        if issues_value == -2 and direction_changes < 2:
			#target unreachable
            if rotation_direction == "pos":
                rotation_direction = "neg"
                direction_changes += 1
                r = -1 #rotation factor to make the rotation negative
            else:
                rotation_direction = "pos"
                direction_changes += 1
                r = 1 #rotation factor to make the rotation positive
            issues_value, target_new_pose = test_issues_point(target, r*rotation_step)
            target.setPose(target_new_pose)

        elif issues_value > 0 and rep < repmax:
			#collision
            RDK.setCollisionActive(COLLISION_OFF)
            if DEBUG:
                is_active = RDK.Command("CollisionActive")
                print(f"collsion active? should be off (0) {is_active}")
                debuglist.append(f"collsion active? should be off (0) {is_active}")

            ROBOT.MoveJ(target.Pose())
            if rotation_direction == "neg":
                r = -1
            elif rotation_direction == "pos":
                r = 1
            issues_value, target_new_pose = test_issues_point(target, r*rotation_step)
            target.setPose(target_new_pose)
            rep += 1

        elif direction_changes >= 2 or rep >= repmax:
            break

        else:
            RDK.ShowMessage(f"Unknown error occured at Hole {idx} while looking for collision free position")
            if DEBUG:
                print(f"Unknown error occured at Hole {idx} while looking for collision free position")
                debuglist.append(f"Unknown error occured at Hole {idx} while looking for collision free position")

    direction_changes = 0
    if issues_value == 0:
        print(f"No issues at Hole {idx}")
        debuglist.append(f"No issues at Hole {idx}")
    elif direction_changes >= 2 or rep >= repmax or s >= 100:
        RDK.ShowMessage(f"No solution found for Hole {idx}", False)
        holes_no_solution.append(idx)
        if DEBUG:
            print(f"No solution found for Hole {idx}")
            debuglist.append(f"No solution found for Hole {idx}")
    else:
        RDK.ShowMessage(f"Unknown error occured at Hole {idx} while looking for collision free position")
        if DEBUG:
            print(f"Unknown error occured at Hole {idx} while looking for collision free position")
            debuglist.append(f"Unknown error occured at Hole {idx} while looking for collision free position")


MAKE_GUI_PROGRAM = True

ROBOT.setFrame(FRAME)
ROBOT.setTool(TOOL)

if RDK.RunMode() == RUNMODE_SIMULATE:
    MAKE_GUI_PROGRAM = True
    # MAKE_GUI_PROGRAM = mbox('Do you want to create a new program? If not, the robot will just move along the targets', 'Yes', 'No')
else:
    # if we run in program generation mode just move the robot
    MAKE_GUI_PROGRAM = False

if MAKE_GUI_PROGRAM:
    RDK.Render(False)  # Faster if we turn render off
    make_targets(csv_file)
else:
    l

RDK.ShowMessage(f"Holes without solution: {holes_no_solution}")

if DEBUG:
    print(f"Holes without solution: {holes_no_solution}")
    debuglist.append(f"Holes without solution: {holes_no_solution}")

    current_time = datetime.datetime.now()
    filename = os.path.splitext(os.path.basename(__file__))
    with open("C:/Users/Laura/Documents/1.Windesheim/Stage/2024/Lectoraat/Deelvragen/2.Targets maken/debugfile.txt", "a") as file:
        file.write("\n\n-----------------------------------------------\n")
        file.write(current_time.strftime("%c"))
        file.write("\n-----------------------------------------------\n")
        for prints in debuglist:
            file.write(prints)
            file.write("\n")
        file.write(holes_no_solution)
        file.write(filename[0])

--- Python program Addmoveshanktoprog ---
from robodk import robolink, robomath

# Connect to RoboDK
RDK = robolink.Robolink()

# Ask the user to select the program to duplicate
orig_prog = RDK.ItemUserPick("Select the program to duplicate", robolink.ITEM_TYPE_PROGRAM)
if not orig_prog.Valid():
    print("No valid program selected.")
    quit()

# Create a new program (a duplicate) with a new name
new_prog_name = "New_" + orig_prog.Name()
new_prog = RDK.AddProgram(new_prog_name)
print("Creating new program:", new_prog.Name())

# Get the number of instructions from the original program
ins_count = orig_prog.InstructionCount()
print("Original program '{}' has {} instructions.".format(orig_prog.Name(), ins_count))

# Iterate over each instruction in the original program
for i in range(ins_count):
    # Retrieve instruction info as a dictionary.
    # Note: Calling setParam(i) with only the index returns the instruction information.
    ins_dict = orig_prog.setParam(i)

    # Try to get the command code string from the instruction dictionary.
    # (Many instructions have a "Code" key that holds the Python command as text.)
    code_line = ins_dict.get("Code", "").strip()
    if not code_line:
        print("Skipping instruction {} because no code is available.".format(i))
        continue

    # Add the instruction to the new program
    print("Adding instruction {}: {}".format(i, code_line))
    new_prog.RunInstruction(code_line, robolink.INSTRUCTION_CALL_PROGRAM)

    # If the instruction contains "FaceTarget" then add two extra moveshank instructions after it.
    if "Face_Target" in code_line:
        print("Detected 'FaceTarget' at instruction {}. Inserting moveshank instructions.".format(i))
        new_prog.RunInstruction('move_shank(20)', robolink.INSTRUCTION_CALL_PROGRAM)
        new_prog.RunInstruction('move_shank(0)', robolink.INSTRUCTION_CALL_PROGRAM)

# Finalize the new program; this applies the modifications
new_prog.Update()
print("New program '{}' created successfully.".format(new_prog.Name()))

--- Python program importerTest ---
# This macro loads CSV target files and places them in RoboDK
# Supported CSV format: X,Y,Z,RX,RY,RZ

# Import required modules
from robodk.robolink import *  # API to communicate with RoboDK
from robodk.robomath import *  # Robot toolbox
from robodk.robodialogs import *
from robodk.robofileio import *
import robodk.robolinkutils as RDKutils

# Start communication with RoboDK
RDK = Robolink()

# Ask the user to select the robot
ROBOT = RDK.ItemUserPick('Select a robot', ITEM_TYPE_ROBOT)

# Check if the user selected a robot
if not ROBOT.Valid():
    quit()

# Get the reference frame and active tool
BASE = ROBOT.Parent()
FRAME = RDK.ItemUserPick('Reference Frame', ITEM_TYPE_FRAME)
FRAMEPOSE = RDKutils.getPoseWrt(FRAME, BASE)  # frame pose wrt robot base
TOOL = ROBOT.getLink(ITEM_TYPE_TOOL)
TOOLPOSE = RDKutils.getPoseWrt(TOOL, TOOL.Parent())  # tool pose wrt robot flange

if not FRAME.Valid() or not TOOL.Valid():
    raise Exception("Select appropriate FRAME and TOOL references")

# Function to convert XYZWPR to a pose
def xyzwpr_to_pose(xyzwpr):
    x, y, z, rx, ry, rz = xyzwpr
    return point_Zaxis_2_pose([x, y, z], [rx, ry, rz])

# Ask user to select the CSV file
csv_file = getOpenFileName(RDK.getParam('PATH_OPENSTATION'))

# Specify file codec
codec = 'utf-8'

# Load CSV target data
def load_targets(strfile):
    csvdata = LoadList(strfile, ',', codec)
    poses = []
    idxs = []
    for i in range(0, len(csvdata)):
        x, y, z, rx, ry, rz = csvdata[i][0:6]
        poses.append(xyzwpr_to_pose([x, y, z, rx, ry, rz]))
        idxs.append(i)
    return poses, idxs

# Create targets in RoboDK and move the robot to each target
def process_targets(strfile):
    poses, idxs = load_targets(strfile)
    program_name = getFileName(strfile)
    program_name = program_name.replace('-', '_').replace(' ', '_')

    # Set the robot's frame and tool
    ROBOT.setFrame(FRAME)
    ROBOT.setTool(TOOL)

    # Create a program to visit all targets
    program = RDK.AddProgram('Visit_' + program_name, ROBOT)

    for pose, idx in zip(poses, idxs):
        # Create target name
        name = 'Target-%s-%i' % (program_name, idx)

        # Delete target if it already exists
        target = RDK.Item(name, ITEM_TYPE_TARGET)
        if target.Valid():
            target.Delete()

        # Create new target
        target = RDK.AddTarget(name, FRAME, ROBOT)
        target.setPose(pose)

        # Add a movement instruction to the program
        program.MoveJ(target)

        # Optional: Move the robot to the target in simulation
        RDK.setSimulationSpeed(1)  # Normal speed
        ROBOT.MoveJ(target)

# Main execution
if __name__ == "__main__":
    # Ask user whether to just create targets or also move the robot
    move_robot = RDK.RunMode() != RUNMODE_SIMULATE

    if move_robot:
        # We're in run mode, just move the robot to targets
        poses, idxs = load_targets(csv_file)
        for pose, idx in zip(poses, idxs):
            ROBOT.MoveJ(pose)
    else:
        # We're in simulation mode, create targets and a program
        process_targets(csv_file)

    RDK.ShowMessage("Target processing complete", False)

--- program Prog20 (robot UR10e) ---
  Set Ref.: CSV Frame
  Set Tool: TCP Schroeftool at (225.74, 0.91, 101.72) mm, rotated rx 90 ry -90 rz 90 deg
  MoveL (Target 36)
  Call Program_Face_-1_0_0
  Call Program_Face_-1_0_0
  MoveL (Target 36)
  MoveL (Target 35)
  MoveJ (Target 37 new)
  MoveL (Target 37 new)
  MoveL (Target 35)
  Call Program_Face_0_-1_1
  MoveL (Target 35)
  Call Program_Face_0_-1_0
  MoveL (Target 35)

--- program Program_Face_-1_0_0 (robot UR10e) ---
  Set Ref.: CSV Frame
  Set Tool: schroevendraaier all in met meet cone (1)
  MoveL (Target 36)
  MoveL (Face_Target_-1_0_0)
  MoveL (H-12.5_30.0-9)
  MoveL (Face_Target_-1_0_0)
  MoveL (H-12.5_30.0-10)
  MoveL (Face_Target_-1_0_0)
  MoveL (H-12.5_30.0-11)
  MoveL (Face_Target_-1_0_0)
  MoveL (H-12.5_30.0-12)
  MoveL (Face_Target_-1_0_0)
  MoveL (H-12.5_30.0-13)
  MoveL (Face_Target_-1_0_0)
  MoveL (H-12.5_30.0-14)
  MoveL (Face_Target_-1_0_0)
  MoveL (H-12.5_30.0-15)
  MoveL (Face_Target_-1_0_0)
  MoveL (Target 36)

--- program Program_Face_0_0_1 (robot UR10e) ---
  Set Ref.: CSV Frame
  Set Tool: schroevendraaier all in met meet cone (1)
  MoveL (Face_Target_0_0_1)
  MoveL (H-12.4_20.0-0)
  MoveL (Face_Target_0_0_1)
  MoveL (H-12.4_20.0-1)
  MoveL (Face_Target_0_0_1)
  MoveL (H-12.4_20.0-2)
  MoveL (Face_Target_0_0_1)
  MoveL (H-12.4_20.0-3)
  MoveL (Face_Target_0_0_1)
  MoveL (H-12.4_20.0-4)
  MoveL (Face_Target_0_0_1)
  MoveL (H-12.4_20.0-5)
  MoveL (Face_Target_0_0_1)
  MoveL (H-12.4_20.0-6)
  MoveL (Face_Target_0_0_1)

--- program Program1hole3sides27May (robot UR10e) ---
  Set Ref.: CSV Frame
  Set Tool: schroevendraaier all in met meet cone (1)
  MoveL (Target 35)
  MoveL (oppak)
  Call screw_in(0)
  MoveL (Target 35)
  MoveL (Face_Target_0_-1_0)
  MoveL (H-8.3_20.0-15)
  Call screw_in(20)
  Call screw_out(0)
  MoveL (Face_Target_0_-1_0)
  MoveL (Target 35)
  MoveL (oppak)
  Call screw_in(0)
  MoveL (Target 35)
  MoveL (Face_Target_0_-1_0)
  MoveL (H-8.3_20.0-16)
  Call screw_in(20)
  Call screw_out(0)
  MoveL (Face_Target_0_-1_0)
  MoveL (Target 35)
  MoveL (oppak)
  Call screw_in(0)
  MoveL (Target 35)
  MoveL (Face_Target_0_-1_0)
  MoveL (H-8.3_20.0-17)
  Call screw_in(20)
  Call screw_out(0)
  MoveL (Face_Target_0_-1_0)
  MoveL (Target 35)
  MoveL (oppak)
  Call screw_in(0)
  MoveL (Target 35)
  MoveL (Face_Target_0_-1_1)
  MoveL (H-8.3_20.0-11)
  Call screw_in(20)
  Call screw_out(0)
  MoveL (Face_Target_0_-1_1)
  MoveL (Target 35)
  MoveL (oppak)
  Call screw_in(0)
  MoveL (Target 35)
  MoveL (Face_Target_0_-1_1)
  MoveL (H-8.3_20.0-13)
  Call screw_in(20)
  Call screw_out(0)
  MoveL (Face_Target_0_-1_1)
  MoveL (Target 35)
  MoveL (oppak)
  Call screw_in(0)
  MoveL (Target 35)
  MoveL (Face_Target_0_-1_1)
  MoveL (H-8.3_20.0-9)
  Call screw_in(20)
  Call screw_out(0)
  MoveL (Face_Target_0_-1_1)
  MoveL (Target 35)
  MoveL (oppak)
  Call screw_in(0)
  MoveL (Target 105)
  MoveL (H-8.3_20.0-2)
  Call screw_in(20)
  Call screw_out(0)
  MoveL (Target 105)
  MoveL (Target 35)
  MoveL (oppak)
  Call screw_in(0)
  MoveL (Target 105)
  MoveL (H-8.3_20.0-1)
  Call screw_in(20)
  Call screw_out(0)
  MoveL (Target 105)
  MoveL (Target 35)
  MoveL (oppak)
  Call screw_in(0)
  MoveL (Target 105)
  MoveL (H-8.3_20.0-3)
  Call screw_in(20)
  Call screw_out(0)
  MoveL (approachvoorkant3)
  MoveL (Target 35)

--- program Program_Face_0_-1_1 (robot UR10e) ---
  Set Ref.: CSV Frame
  Set Tool: schroevendraaier all in met meet cone (1)
  MoveL (Target 35)
  MoveJ (Target 37 new)
  MoveL (Toolswitch-m8)
  Call move_shank(20)
  Call move_shank(0)
  MoveL (Aanlevering-Pos1)
  Call move_shank(20)
  Call move_shank(0)
  MoveJ (Target 37 new)
  MoveJ (Target 35)
  MoveL (Face_Target_0_-1_1)
  MoveL (H-12.4_20.0-10)
  Call move_shank(20)
  Call move_shank(0)
  MoveL (Target 35)
  MoveJ (Target 37 new)
  MoveL (Aanlevering-Pos1)
  Call move_shank(20)
  Call move_shank(0)
  MoveJ (Target 37 new)
  MoveJ (Target 35)
  MoveL (Face_Target_0_-1_1)
  MoveL (H-12.4_20.0-11)
  Call move_shank(20)
  Call move_shank(0)
  MoveL (Target 35)
  MoveJ (Target 37 new)
  MoveL (Aanlevering-Pos1)
  Call move_shank(20)
  Call move_shank(0)
  MoveJ (Target 37 new)
  MoveJ (Target 35)
  MoveL (Face_Target_0_-1_1)
  MoveL (H-12.4_20.0-12)
  Call move_shank(20)
  Call move_shank(0)
  MoveL (Target 35)
  MoveJ (Target 37 new)
  MoveL (Aanlevering-Pos1)
  Call move_shank(20)
  Call move_shank(0)
  MoveJ (Target 37 new)
  MoveJ (Target 35)
  MoveL (Face_Target_0_-1_1)
  MoveL (H-12.4_20.0-13)
  Call move_shank(20)
  Call move_shank(0)
  MoveL (Target 35)
  MoveJ (Target 37 new)
  MoveL (Aanlevering-Pos1)
  Call move_shank(20)
  Call move_shank(0)
  MoveJ (Target 37 new)
  MoveJ (Target 35)
  MoveL (Face_Target_0_-1_1)
  MoveL (H-12.4_20.0-14)
  Call move_shank(20)
  Call move_shank(0)
  MoveL (Target 35)
  MoveJ (Target 37 new)
  MoveL (Aanlevering-Pos1)
  Call move_shank(20)
  Call move_shank(0)
  MoveJ (Target 37 new)
  MoveL (Target 35)
  - Wanneer face target wordt gemaakt, tussen elke gat moet een helicoil opgepakt worden
- manier bedenken om "Aanlevering-Pos1" target te zoeken 
- manier om Toolswitch-m8 target te zoeken
- wanneer de aanlevering of toolswitch benadert wordt moet dat via target 35 -> target 37

wat er nu aangepast moet worden, moet via de approach points benaderd worden 
de flow voor een gat is de volgende Target 35 -> Target 37 -> Oppakken helicoil, dan via hetzelfde route terug gaan, Target 37 -> Target 35 en naar approach. 
voor elke gat moeten er minimaal 5 bewegingen komen

--- program Program_Face_0_-1_1_m8 (robot UR10e) ---
  Set Ref.: CSV Frame
  Set Tool: TCP Schroeftool at (225.74, 0.91, 101.72) mm, rotated rx 90 ry -90 rz 90 deg
  MoveL (Target 35)
  MoveJ (Target 37 new)
  MoveL (Toolswitch-m8)
  Call move_shank(20)
  Call move_shank(0)
  MoveL (Aanlevering-Pos1)
  Call move_shank(20)
  Call move_shank(0)
  MoveJ (Target 37 new)
  MoveJ (Target 35)
  MoveJ (Target 37 new)
  MoveL (Aanlevering-Pos1)
  Call move_shank(20)
  Call move_shank(0)
  MoveJ (Target 37 new)
  MoveJ (Target 35)
  MoveL (Face_Target_0_-1_1)
  MoveL (H-8.3_20.0-8)
  Call move_shank(20)
  Call move_shank(0)
  MoveL (Target 35)
  MoveJ (Target 37 new)
  MoveL (Aanlevering-Pos1)
  Call move_shank(20)
  Call move_shank(0)
  MoveJ (Target 37 new)
  MoveJ (Target 35)
  MoveL (Face_Target_0_-1_1)
  MoveL (H-8.3_20.0-9)
  Call move_shank(20)
  Call move_shank(0)
  MoveL (Target 35)
  MoveJ (Target 37 new)
  MoveL (Aanlevering-Pos1)
  Call move_shank(20)
  Call move_shank(0)
  MoveJ (Target 37 new)
  MoveJ (Target 35)
  MoveL (Face_Target_0_-1_1)
  MoveL (H-8.3_20.0-10)
  Call move_shank(20)
  Call move_shank(0)
  MoveL (Target 35)
  MoveJ (Target 37 new)
  MoveL (Aanlevering-Pos1)
  Call move_shank(20)
  Call move_shank(0)
  MoveJ (Target 37 new)
  MoveJ (Target 35)
  MoveL (Face_Target_0_-1_1)
  MoveL (H-8.3_20.0-11)
  Call move_shank(20)
  Call move_shank(0)
  MoveL (Target 35)
  MoveJ (Target 37 new)
  MoveL (Aanlevering-Pos1)
  Call move_shank(20)
  Call move_shank(0)
  MoveJ (Target 37 new)
  MoveL (Target 35)
  MoveJ (Target 37 new)
  MoveL (Aanlevering-Pos1)
  Call move_shank(20)
  Call move_shank(0)
  MoveJ (Target 37 new)
  MoveJ (Target 35)
  MoveL (Face_Target_0_-1_1)
  MoveL (H-8.3_20.0-12)
  Call move_shank(20)
  Call move_shank(0)
  MoveL (Target 35)
  MoveJ (Target 37 new)
  MoveL (Aanlevering-Pos1)
  Call move_shank(20)
  Call move_shank(0)
  MoveJ (Target 37 new)
  MoveJ (Target 35)
  MoveL (Face_Target_0_-1_1)
  MoveL (H-8.3_20.0-13)
  Call move_shank(20)
  Call move_shank(0)
  MoveL (Target 35)
  - Wanneer face target wordt gemaakt, tussen elke gat moet een helicoil opgepakt worden
- manier bedenken om "Aanlevering-Pos1" target te zoeken 
- manier om Toolswitch-m8 target te zoeken
- wanneer de aanlevering of toolswitch benadert wordt moet dat via target 35 -> target 37

wat er nu aangepast moet worden, moet via de approach points benaderd worden 
de flow voor een gat is de volgende Target 35 -> Target 37 -> Oppakken helicoil, dan via hetzelfde route terug gaan, Target 37 -> Target 35 en naar approach. 
voor elke gat moeten er minimaal 5 bewegingen komen

--- program Program_Face_0_-1_0 (robot UR10e) ---
  Set Ref.: CSV Frame
  Set Tool: TCP Schroeftool at (225.74, 0.91, 101.72) mm, rotated rx 90 ry -90 rz 90 deg
  MoveL (Face_Target_0_-1_0)
  MoveL (H-12.4_20.0-18)
  MoveL (Face_Target_0_-1_0)
  MoveL (H-12.4_20.0-19)
  MoveL (Face_Target_0_-1_0)
  MoveL (H-12.4_20.0-20)
  MoveL (Face_Target_0_-1_0)
  MoveL (H-12.4_20.0-21)
  MoveL (Face_Target_0_-1_0)
  MoveL (H-12.4_20.0-22)
  MoveL (Face_Target_0_-1_0)

--- program Prog22 (robot UR10e) ---
  Set Ref.: CSV Frame
  Set Tool: TCP Schroeftool at (225.74, 0.91, 101.72) mm, rotated rx 90 ry -90 rz 90 deg
  MoveL (Target 36)
  MoveL (Target 35)
  MoveJ (Target 37 new)
  MoveL (Toolswitch-m8)
  Call move_shank(20)
  Call move_shank(0)
  MoveL (H-10.2_4-0) -> target Aanlevering-Pos1
  Call move_shank(20)
  Call move_shank(0)
  MoveL (Target 37 new)

--- program Visit_8.3_20.0 (robot UR10e) ---
  MoveJ (Target-8.3_20.0-0) [its target is no longer in the station]

--- program Visit_8.3_20.0 (robot UR10e) ---
  MoveJ (Target-8.3_20.0-0) [its target is no longer in the station]
  MoveJ (Target-8.3_20.0-1) [its target is no longer in the station]
  MoveJ (Target-8.3_20.0-2) [its target is no longer in the station]
  MoveJ (Target-8.3_20.0-3) [its target is no longer in the station]
  MoveJ (Target-8.3_20.0-4) [its target is no longer in the station]
  MoveJ (Target-8.3_20.0-5) [its target is no longer in the station]
  MoveJ (Target-8.3_20.0-6) [its target is no longer in the station]
  MoveJ (Target-8.3_20.0-7) [its target is no longer in the station]
  MoveJ (Target-8.3_20.0-8) [its target is no longer in the station]
  MoveJ (Target-8.3_20.0-9) [its target is no longer in the station]
  MoveJ (Target-8.3_20.0-10) [its target is no longer in the station]
  MoveJ (Target-8.3_20.0-11) [its target is no longer in the station]
  MoveJ (Target-8.3_20.0-12) [its target is no longer in the station]
  MoveJ (Target-8.3_20.0-13) [its target is no longer in the station]
  MoveJ (Target-8.3_20.0-14) [its target is no longer in the station]
  MoveJ (Target-8.3_20.0-15) [its target is no longer in the station]

--- program Visit_8.3_20.0 (robot UR10e) ---
  MoveJ (Target-8.3_20.0-0) [its target is no longer in the station]
  MoveJ (Target-8.3_20.0-1) [its target is no longer in the station]
  MoveJ (Target-8.3_20.0-2) [its target is no longer in the station]
  MoveJ (Target-8.3_20.0-3) [its target is no longer in the station]
  MoveJ (Target-8.3_20.0-4) [its target is no longer in the station]
  MoveJ (Target-8.3_20.0-5) [its target is no longer in the station]
  MoveJ (Target-8.3_20.0-6) [its target is no longer in the station]
  MoveJ (Target-8.3_20.0-7) [its target is no longer in the station]
  MoveJ (Target-8.3_20.0-8) [its target is no longer in the station]
  MoveJ (Target-8.3_20.0-9) [its target is no longer in the station]
  MoveJ (Target-8.3_20.0-10) [its target is no longer in the station]
  MoveJ (Target-8.3_20.0-11) [its target is no longer in the station]
  MoveJ (Target-8.3_20.0-12) [its target is no longer in the station]
  MoveJ (Target-8.3_20.0-13) [its target is no longer in the station]
  MoveJ (Target-8.3_20.0-14) [its target is no longer in the station]
  MoveJ (Target-8.3_20.0-15) [its target is no longer in the station]
  MoveJ (Target-8.3_20.0-16) [its target is no longer in the station]
  MoveJ (Target-8.3_20.0-17) [its target is no longer in the station]
  MoveJ (Target-8.3_20.0-18) [its target is no longer in the station]

--- program Prog28 (robot UR10e) ---
  Set Ref.: CSV Frame
  Set Tool: TCP Schroeftool at (225.74, 0.91, 101.72) mm, rotated rx 90 ry -90 rz 90 deg
  MoveL (Target 93)
  MoveL (Target 94)
  MoveL (H-8.3_20.0-0)

--- program Prog29 (robot UR10e) ---
  Set Ref.: CSV Frame
  Set Tool: schroevendraaier all in met meet cone (1)
  MoveJ (Target 37 new)
  MoveL (oppak)
  Call screw_in(20)
  MoveJ (Target 37 new)
  MoveL (Target 35)
  MoveL (Face_Target_0_-1_1)
  MoveL (H-8.3_20.0-9)
  Call screw_in(20)
  Call screw_out(20)
  MoveL (Target 35)
  Call Program1
  MoveJ (Target 37 new)
  MoveL (oppak)
  Call screw_in(20)
  MoveJ (Target 37 new)
  MoveL (Target 35)
  MoveL (Face_Target_0_-1_1)
  MoveL (H-8.3_20.0-13)
  Call screw_in(20)
  Call screw_out(20)
  MoveL (Target 35)
  Call Program1

--- program Prog30 (robot UR10e) ---
  Set Ref.: CSV Frame
  Set Tool: schroevendraaier all in met meet cone (1)
  MoveL (H-8.3_20.0-17)
  MoveL (H-8.3_20.0-18)
  MoveL (H-8.3_20.0-15)
  MoveL (H-8.3_20.0-14)

--- program voorkant3gaten (robot UR10e) ---
  Set Ref.: CSV Frame
  Set Tool: schroevendraaier all in met meet cone (1)
  MoveL (Target 35)
  MoveL (oppak)
  Call screw_in(0)
  MoveL (Target 105)
  MoveL (H-8.3_20.0-2)
  Call screw_in(20)
  Call screw_out(0)
  MoveL (Target 105)
  MoveL (Target 35)
  MoveL (oppak)
  Call screw_in(0)
  MoveL (Target 105)
  MoveL (H-8.3_20.0-1)
  Call screw_in(20)
  Call screw_out(0)
  MoveL (Target 105)
  MoveL (Target 35)
  MoveL (oppak)
  Call screw_in(0)
  MoveL (Target 105)
  MoveL (H-8.3_20.0-3)
  Call screw_in(20)
  Call screw_out(0)
  MoveL (Target 35)

--- program Prog30-schuin (robot UR10e) ---
  Set Ref.: CSV Frame
  Set Tool: schroevendraaier all in met meet cone (1)
  MoveL (H-8.3_20.0-10)
  MoveL (H-8.3_20.0-11)
  MoveL (H-8.3_20.0-12)

--- program Prog30-voorkant (robot UR10e) ---
  Set Ref.: CSV Frame
  Set Tool: schroevendraaier all in met meet cone (1)
  MoveL (H-8.3_20.0-3)
  MoveL (H-8.3_20.0-4)
  MoveL (H-8.3_20.0-0)
  MoveL (H-8.3_20.0-1)
  MoveL (H-8.3_20.0-5)

--- Python program Create measurements 3DOF ---
# type help("robolink") or help("robodk") for more information
# (note: you do not need to keep a copy of this file, your python script is saved with the station)
from robodk.robolink import *  # API to communicate with robodk
from robodk.robomath import *  # basic matrix operations
from robodk.robodialogs import *
from random import uniform
import sys  # to exit the script without errors (sys.exit(0))
import re  # to convert a string list into a list of values


def CreateMeasurementsPoint(calib_targets=None):

    DEFAULT_NMEASURES = 80
    # Default limit space in the Cartesian space
    DEFAULT_XYZ_MIN = [-5000, -5000, 0]
    DEFAULT_XYZ_MAX = [5000, 5000, 5000]

    TRACKER_REF_NAME = 'Tracker Reference'  # keyword of the measurement system reference (in RoboDK)
    TCP_PREFIX = 'CalibTool'

    # Use the tag CHECK_COLLISION_NAME to automatically turn the objects visible. This will allow to detect collisions.
    CHECK_COLLISION = True
    CHECK_COLLISION_MOVE = True
    CHECK_COLLISION_NAME = 'collision'
    CHECK_COLLISION_STEP = -1  # in degrees, step to check for collisions. higher is faster.

    # Use the tag CHECK_COLLISION_NAME to automatically turn the objects visible. This will allow to detect collisions.
    CHECK_WORKSPACE = False
    CHECK_WORKSPACE_NAME = 'Workspace'

    # Avoid a cylinder located at X=0, Y=0 or radius R_MIN
    R_MIN = 100
    R_MIN_Z = 200

    # Allow rotations of the tool pointing to the measurement system
    ROTX_MIN = -5
    ROTX_MAX = 5
    ROTY_MIN = -5
    ROTY_MAX = 5
    ROTZ_MIN = -180
    ROTZ_MAX = 180

    # use FILE_SAVE_PREFIX to automatically save the file, otherwise, comment this line
    # FILE_SAVE_PREFIX = 'CalibrationSequence'

    # --------------------------------------------------------------
    def to_list(str_values, expected_values):
        """Converts a string into a list of values. It returns None if the array is smaller than the expected size."""
        if str_values is None:
            return None
        values = re.findall("[-+]?\d+[\.]?\d*", str_values)
        if len(values) < expected_values:
            return None
        for i in range(len(values)):
            values[i] = float(values[i])
        print('Read values: ' + repr(values))
        return values

    def get_values(title_msg, show_value, expected_values):
        """Gets a list of values from the user, stops the script if the user hits cancel"""
        if type(show_value) == Mat:
            show_value = show_value.tolist()
        answer = mbox(title_msg, entry=str(show_value))
        if answer is False:
            print('Operation cancelled by user')
            sys.exit(0)
            #raise Exception('Operation cancelled by user')
        #print('Input value: ' + answer)
        values = to_list(answer, expected_values)
        #if len(values) < expected_values:
        #    raise Exception('%i values expected' % expected_values)
        return values

    def stop_script():
        """Forces the script to finish with/without errors"""
        # raise Exception('Operation cancelled by user')
        print('Operation cancelled by user')
        sys.exit(0)

    # ---------------------------------
    RDK = Robolink()

    # Disable collision checking (otherwise, the program stops)
    RDK.setCollisionActive(COLLISION_OFF)

    # get previously set variables
    NMEASURES = RDK.getParam('CALIB_MEASUREMENTS')
    #JOINTS_REF = to_list(RDK.getParam('CALIB_JOINTS_REF'), 6)
    ANG_MIN = to_list(RDK.getParam('CALIB_JOINTLIM_LOW'), 6)
    ANG_MAX = to_list(RDK.getParam('CALIB_JOINTLIM_HIGH'), 6)
    XYZ_MIN = to_list(RDK.getParam('CALIB_XYZLIM_LOW'), 3)
    XYZ_MAX = to_list(RDK.getParam('CALIB_XYZLIM_HIGH'), 3)

    INPUT_VALUES = False
    # force user input if one of the variables is not set
    if NMEASURES is None or ANG_MIN is None or ANG_MAX is None:  # or XYZ_MIN is None or XYZ_MAX is None:
        INPUT_VALUES = True

    #----------------------- Select robot ------------------
    robot = RDK.ItemUserPick("Select a robot for calibration/validation", ITEM_TYPE_ROBOT)
    if not robot.Valid():
        raise Exception('Robot not selected or no robot available')
    print('Using robot: %s' % robot.Name())
    #------------------------------------------------------------

    #----------------------- Select tracker ------------------
    tracker = RDK.Item(TRACKER_REF_NAME)
    if not tracker.Valid():
        frame_ref = RDK.AddFrame('Measurements Reference', robot.Parent())
        frame_ref.setPose(transl(2000, 0, 1000))
        tracker = RDK.AddFrame(TRACKER_REF_NAME, frame_ref)
        tracker.setPose(transl(0, 0, 0))
        tracker.setVisible(False)
    #    tracker = RDK.ItemUserPick('Select the measurement system reference:<br>(avoid this message by naming the tracker reference "%s")' % TRACKER_REF_NAME, ITEM_TYPE_FRAME)
    #    if not tracker.Valid():
    #        stop_script()

    #----------------------- Select tool and workspace object to verify if tool is inside the object
    tool_object = None
    workspace_object = None
    if CHECK_WORKSPACE:
        # tool_object is the geometry of the tool used to check if the tool is inside the workspace
        robot_tools = robot.Childs()
        for tooli in robot_tools:
            if tooli.Name().find(CHECK_COLLISION_NAME) >= 0:
                tool_object = tooli
        if tool_object is None and len(robot_tools) > 0:
            tool_object = robot_tools[0]

        # workspace object is the workspace of the tracker (object)
        workspace_object = RDK.Item(CHECK_WORKSPACE_NAME, ITEM_TYPE_OBJECT)
    #------------------------------------------------------------

    #if JOINTS_REF is None:
    #    # Use robot home position as default reference joints
    #    JOINTS_REF = robot.JointsHome().tolist()

    if XYZ_MIN is None:
        XYZ_MIN = DEFAULT_XYZ_MIN

    if XYZ_MAX is None:
        XYZ_MAX = DEFAULT_XYZ_MAX

    [ang_min_robot, ang_max_robot, JOINTS_TYPE] = robot.JointLimits()
    if ANG_MIN is None or ANG_MAX is None:
        ANG_MIN = ang_min_robot.tolist()
        ANG_MAX = ang_max_robot.tolist()
        # limit joint axes from -180 to +180 (no need to go farther for calibration)
        for i in [3, 5]:
            ANG_MIN[i] = max(ANG_MIN[i], -180)
            ANG_MAX[i] = min(ANG_MAX[i], 180)

        ANG_MIN[0] = max(ANG_MIN[0], -90)
        ANG_MAX[0] = min(ANG_MAX[0], 90)

        ANG_MIN[4] = max(ANG_MIN[4], -90)
        ANG_MAX[4] = min(ANG_MAX[4], 90)

        print('Using default robot joint limits:')
        print(ANG_MIN)
        print(ANG_MAX)

    while True:
        # Loop until the user inputs variables that are accepted
        if INPUT_VALUES:
            # Ask the user to validate/enter all the settings

            # ---------------- getting the number of measurements
            if NMEASURES is None or type(NMEASURES) == str:
                NMEASURES = DEFAULT_NMEASURES
            input_val = mbox('Enter the number of measurements:\n(at least 60 measurements are recommended for robot calibration)', entry=str(NMEASURES))
            if input_val is False:
                stop_script()

            NMEASURES = int(float(input_val))
            RDK.setParam('CALIB_MEASUREMENTS', NMEASURES)

            # ---------------- getting the Reference Joints
            #robot.setJoints(JOINTS_REF)
            #answer = mbox('Set the robot reference joints and select OK. The tool must be facing the tracker for this position.\nCurrent values: %s' % str(JOINTS_REF))
            #if answer is False:
            #    stop_script()

            #JOINTS_REF = robot.Joints().tolist()
            #RDK.setParam('CALIB_JOINTS_REF', JOINTS_REF)

            # ---------------- getting the Joint limits (lower bound)
            robot.setJoints(ANG_MIN)
            answer = mbox('Set the Joint limits (LOWER bound, in deg), then select OK.\nCurrent values: %s' % str(ANG_MIN))
            if answer is False:
                stop_script()

            ANG_MIN = robot.Joints().tolist()
            RDK.setParam('CALIB_JOINTLIM_LOW', ANG_MIN)

            # ---------------- getting the Joint limits (upper bound)
            robot.setJoints(ANG_MAX)
            answer = mbox('Set the Joint limits (UPPER bound, in deg), then select OK.\nCurrent values: %s' % str(ANG_MAX))
            if answer is False:
                stop_script()

            ANG_MAX = robot.Joints().tolist()
            RDK.setParam('CALIB_JOINTLIM_HIGH', ANG_MAX)

            # ---------------- getting the XYZ limits (lower bound)
            #XYZ_MIN = get_values('Enter the Cartesian limits (lower bound, in mm), then select OK.', XYZ_MIN, 3)
            #RDK.setParam('CALIB_XYZLIM_LOW', XYZ_MIN)

            # ---------------- getting the XYZ limits (upper bound)
            #XYZ_MAX = get_values('Enter the Cartesian limits (upper bound, in mm), then select OK.', XYZ_MAX, 3)
            #RDK.setParam('CALIB_XYZLIM_HIGH', XYZ_MAX)

        # show summary of parameters
        #robot.setJoints(JOINTS_REF)
        summary_msg = 'Current settings to generate robot calibration configurations:\n\n'
        summary_msg += ('Number of points: %i\n' % NMEASURES)
        #summary_msg += ('Reference joints (deg): %s\n' % str([ round(elem) for elem in JOINTS_REF ]))
        summary_msg += ('Tracker object: %s\n' % tracker.Name())
        if tool_object is not None and workspace_object is not None and workspace_object.Valid() and workspace_object.Visible():
            CHECK_WORKSPACE = True
            summary_msg += ('Creating targets inside tracker workspace (hide workspace to deactivate)\n\n')
        else:
            CHECK_WORKSPACE = False
            summary_msg += ('Skip creating targets inside the tracker workspace (show workspace to activate)\n\n')
        summary_msg += ('Lower joint limits (deg): %s\n' % str(ANG_MIN))
        summary_msg += ('Upper joint limits (deg): %s\n\n' % str(ANG_MAX))
        summary_msg += ('Lower Cartesian limits (mm): %s\n' % str(XYZ_MIN))
        summary_msg += ('Upper Cartesian limits (mm): %s\n\n' % str(XYZ_MAX))
        summary_msg += ('Important: Define collision map settings to check for collisions (select: Tools->Collision Map)\n\n')
        summary_msg += ('Continue?')

        answer = mbox(summary_msg, b1=('Start', 's'), b2=('Edit', 'e'))
        pause(0.001)  # Make tkinter disappear on Mac
        if answer == 'e':
            # Continue loop until the summary is accepted
            INPUT_VALUES = True
            continue

        # if paramters are OK, exit the loop and continue
        break

    # raise Exception('done')

    NDOFS = min(len(robot.Joints().list()), len(ANG_MAX))

    # -----------------------------------------------------
    # Custom-made procedures
    def randjoints():
        """Returns a random set of robot joints within the joint limits."""
        angrand = Mat(NDOFS, 1)
        for i in range(NDOFS):
            angrand[i, :] = uniform(ANG_MIN[i], ANG_MAX[i])
        #jrand = angles_2_joints(angrand.tolist(), JOINTS_TYPE)
        jrand = angrand.tolist()
        return Mat(jrand)

    def check_joints(jin):
        """Returns true if the joints are within the accepted limits."""
        if not isinstance(jin, Mat):
            return False
        if jin.size(0) < 6:
            return False
        #angles = joints_2_angles(jin.tolist(), JOINTS_TYPE)
        angles = jin.tolist()
        for i in range(NDOFS):
            if angles[i] > ANG_MAX[i] or angles[i] < ANG_MIN[i]:
                print("        Joint %i out of limits (%.1f)" % ((i + 1), angles[i]))
                return False
        return True

    def check_pose(hin):
        """Returns true if the pose is within the accepted limits."""
        x = hin[0, 3]
        y = hin[1, 3]
        z = hin[2, 3]
        if x < XYZ_MIN[0] or x > XYZ_MAX[0]:
            print("        X coordinate out of limits %.1f" % x)
        elif y < XYZ_MIN[1] or y > XYZ_MAX[1]:
            print("        Y coordinate out of limits %.1f" % y)
        elif z < XYZ_MIN[2] or z > XYZ_MAX[2]:
            print("        Z coordinate out of limits %.1f" % z)
        elif x * x + y * y < R_MIN * R_MIN and z < R_MIN_Z:
            print("        Robot wrist too close to the robot")
        else:
            return True
        return False

    def randpose(rob, htool, point):
        """Returns a random pose where the Z axis points to the measurement system within the accepted rotation limits.
        The point must be given with respect to the robot reference frame."""
        while True:
            jrand = randjoints()
            try:
                print("Random joints: " + str(jrand.list()))
                hrand = rob.SolveFK(jrand) * htool
            except:
                continue
            prand = hrand[0:3, 3].tolist()
            zvect = normalize3(subs3(point, prand))
            xaprox = [0, 0, 1]
            if angle3(zvect, xaprox) < 5 * pi / 180:
                xaprox = [0, 1, 0]
            yvect = normalize3(cross(zvect, xaprox))
            xvect = cross(yvect, zvect)
            hrand[0:3, 0] = xvect
            hrand[0:3, 1] = yvect
            hrand[0:3, 2] = zvect
            rx = uniform(ROTX_MIN, ROTX_MAX) * pi / 180
            ry = uniform(ROTY_MIN, ROTY_MAX) * pi / 180
            rz = uniform(ROTZ_MIN, ROTZ_MAX) * pi / 180
            hrand = hrand * rotx(rx) * roty(ry) * rotz(rz)
            return hrand

    # -------------------------------------------------------------
    # Program start:

    # Get the robot tool list
    tools = robot.Childs()

    # Get tools to calibrate (tools nambed with TCP_PREFIX):
    # Also, set visible the tools named with CHECK_COLLISION_NAME to check collisions

    sethidden = []
    print('Robot tools:')
    Htools = []
    ntools = len(tools)
    for i in range(ntools):
        tooli = tools[i]
        tooli_name = tooli.Name()
        if tooli_name.find(TCP_PREFIX) == 0:
            Htooli = tooli.PoseTool()
            print('Using %s to calibrate' % tooli_name)
            print(Htooli)
            Htools.append(Htooli)
        if tooli_name.find(CHECK_COLLISION_NAME) >= 0:
            print('Using TCP %s to check collision' % tooli_name)
            # Set the tool visible and remember if it was invisible to turn it off
            if not tooli.Visible():
                sethidden.append(tooli)
                tooli.setVisible(True)

    # Get objects to check collisions:
    all_objects = RDK.ItemList(ITEM_TYPE_OBJECT, True)
    nobjects = len(all_objects)
    for i in range(nobjects):
        objecti = RDK.Item(all_objects[i])
        objecti_name = objecti.Name()
        if objecti_name.find(CHECK_COLLISION_NAME) >= 0:
            print('Using object %s to check collision' % objecti_name)
            # Set the object visible and remember if it was hidden to turn it off
            if not objecti.Visible():
                sethidden.append(objecti)
                objecti.setVisible(True)

    ntools = len(Htools)
    if ntools <= 0:
        tooli = robot.AddTool(transl(100, 0, 100), TCP_PREFIX + ' 1')
        Htools.append(tooli.PoseTool())
        ntools = len(Htools)
        # raise Exception('No tools found with prefix: ' + TCP_PREFIX + '.\nRename the tools that you need to calibrate with the prefix: ' + TCP_PREFIX)

    Htracker_wrt_robot = invH(robot.PoseAbs()) * tracker.PoseAbs()
    ptracker = Htracker_wrt_robot[0:3, 3].tolist()

    # -----------------------------------------------------------------------
    print('Generating ' + repr(NMEASURES) + ' calibration/validation measurements.')
    JLIST = Mat(6, 0)
    JOINTS_REF = robot.JointsHome()

    #-----------
    robot.setJoints(JOINTS_REF)
    while CHECK_COLLISION and RDK.Collisions():
        RDK.Render()
        if ShowMessageYesNoCancel("The robot is in a collision state for the reference joints. Move the robot away from collisions.\n\nContinue?") is True:
            continue
        RDK.setCollisionActive(COLLISION_ON)
        quit()
    RDK.setCollisionActive(COLLISION_OFF)
    #-----------

    JOINTS_REF = robot.Joints()

    LAST_JOINTS = JOINTS_REF  #robot.Joints()
    TCPLIST = Mat(3, 0)

    i = -1
    id_measure = 0
    timeused = 0
    timeleft = -1
    tic()

    while id_measure < NMEASURES:
        i = i + 1
        idtool = id_measure % ntools
        Htool = Htools[idtool]
        ptool = Htool[0:3, 3]
        iHtool = invH(Htool)
        hi = randpose(robot, Htool, ptracker)
        print('Nmeasures: ' + repr(id_measure))
        print('Iteration: ' + repr(i))
        pose_flange = hi * iHtool
        print(pose_flange)
        ji = robot.SolveIK(pose_flange, JOINTS_REF)
        print('Testing Joints: ' + str(ji.list()))
        if not check_joints(ji):
            print('    Joint outside limits')
            continue
        if not check_pose(pose_flange):  #check_pose(hi):
            print('    Pose outside limits')
            continue

        # display potentially good configuration
        robot.setJoints(ji)
        if CHECK_COLLISION and RDK.Collisions():
            print('    End point is in a collision state %i' % i)
            continue
        if CHECK_WORKSPACE and not tool_object.IsInside(workspace_object):
            print('    Tool object outside measurement workspace %i' % i)
            continue
        if CHECK_COLLISION_MOVE and robot.MoveJ_Test(LAST_JOINTS, ji, CHECK_COLLISION_STEP) > 0:
            print('    MoveJ causes collision %i' % i)
            continue

        # robot.setJoints(ji) #this is made automatically by MoveJ_Collision
        LAST_JOINTS = ji
        JLIST = catH(JLIST, ji)
        TCPLIST = catH(TCPLIST, ptool)
        id_measure = id_measure + 1

        # Calculate time
        timeused = toc()
        timeavg = timeused / id_measure
        timeleft = (NMEASURES - id_measure) * timeavg
        print('Elapsed time      : %.1f sec ' % timeused)
        #print('Expected time left: %.1f sec  (average time x measure: %.1f sec)' % (timeleft, timeavg))
        message = 'Calculating measurement configurations. Expected time left: %.1f sec  (found %i/%i measurements)' % (timeleft, id_measure, NMEASURES)
        print(message)
        RDK.ShowMessage(message, False)

    NMEASURES_OK = id_measure
    SAVE_MAT = catV(JLIST, TCPLIST)

    if 'FILE_SAVE_PREFIX' in locals():
        strsave = RDK.getParam('PATH_OPENSTATION') + '/' + FILE_SAVE_PREFIX + repr(NMEASURES_OK) + '.txt'
        SAVE_MAT.save(strsave)
    #else:
    #    strsave = getSaveFile(RDK.getParam('PATH_OPENSTATION'))
    #    strsave = strsave.name
    #    SAVE_MAT.save(strsave)

    # -----------------------------------------------------------------------
    print(tr(JLIST))
    robot.ShowSequence(JLIST)
    RDK.ShowMessage('Calibration/validation sequence found', False)

    # Hide objects that we used to check collisions:
    nhide = len(sethidden)
    for i in range(nhide):
        sethidden[i].setVisible(False)

    # -----------------------------------------------------------------------
    calibitem = RDK.ItemUserPick("Select the calibration project", ITEM_TYPE_CALIBPROJECT)
    if not calibitem.Valid():
        raise Exception("No calibration project selected or available")
        return False

    if calib_targets is None:
        value = mbox('Do you want to use these targets for calibration or validation?', ('Calibration', 'CALIB_TARGETS'), ('Validation', 'VALID_TARGETS'))
    elif calib_targets:
        value = "CALIB_TARGETS"
    else:
        value = "VALID_TARGETS"

    calibitem.setValue(value, SAVE_MAT)

    RDK.ShowMessage('Done', False)

    #mbox('Done')
    # -----------------------------------------------------------------------

    #RDK.ShowSequence(Mat([[1, 10 ,10 ,10 ,10 ,10 ,10],[ 2, 20 ,20 ,20 ,20 ,20 ,20]]))
    return True


if __name__ == "__main__":
    CreateMeasurementsPoint()

--- program Prog34 (robot UR10e) ---
  Set Ref.: CSV Frame
  Set Tool: schroevendraaier all in met meet cone (1)
  MoveL (H-8.3_20.0-8)
  MoveL (H-8.3_20.0-9)
  MoveL (H-8.3_20.0-10)
  MoveL (H-8.3_20.0-11)
  MoveL (H-8.3_20.0-12)
  MoveL (H-8.3_20.0-13)

--- program Prog29-alle zijde 1 (robot UR10e) ---
  Set Ref.: CSV Frame
  Set Tool: schroevendraaier all in met meet cone (1)
  MoveL (Target 37 new)
  MoveL (oppak)
  Call screw_in(0)
  MoveJ (Target 37 new)
  MoveL (Target 35)
  MoveL (Face_Target_0_-1_1)
  MoveL (H-8.3_20.0-9)
  Call screw_in(20)
  Call screw_out(20)
  MoveL (Target 35)
  MoveJ (Target 37 new)
  MoveL (oppak)
  Call screw_in(0)
  MoveJ (Target 37 new)
  MoveL (Target 35)
  MoveL (Face_Target_0_-1_1)
  MoveL (H-8.3_20.0-13)
  Call screw_in(20)
  Call screw_out(20)
  MoveL (Target 35)
  Call Program1
